// TIA Portal project "SCADA_project" (V15.1)

(* hardware
DEVICE "S7300/ET200M station_1"  S7-300 station
   slot 0: "Rail_0"  Rail  6ES7 390-1***0-0AA0
   slot 1: "PS 307 10A_1"  PS 307 10A  6ES7 307-1KA02-0AA0
   slot 2: "PLC_1"  CPU 315-2 PN/DP  6ES7 315-2EH14-0AB0  V3.2
      slot 2: "PROFINET interface_1"  PN-IO
         slot 1: "Port_1"  Port
         slot 2: "Port_2"  Port
   slot 4: "DI 16x24VDC_1"  DI16 x 24VDC  6ES7 321-1BH02-0AA0
   slot 5: "DO 16x24VDC/0.5A_1"  DO16 x 24VDC / 0.5A  6ES7 322-1BH01-0AA0
   slot 6: "AI 8x16BIT_1"  AI8 x 16 bits  6ES7 331-7NF00-0AB0
DEVICE "PC-System_2"  SIMATIC PC station
   slot 0: "SIMATIC PC station"  Rail  SIMATIC PC-Station  V1.0
      slot 125: "Stationmanager"  Station_Manager  V6.0.4
   slot 1: "HMI_RT_2"  WinCC RT Advanced  6AV2 104-0xxxx-xxxx  15.1.0.0
      slot 33792: "Host interface"  Host interface
   slot 2: "IE general_1"  IE General  IE_CP  V8.2.0
*)

// ===== PLC "PLC_1"  CPU 315-2 PN/DP =====

VAR_GLOBAL   // PLC tag table "Default tag table"
   "LT140" AT %ID0 : Real;   // Level transmitter T140
   "LT150" AT %ID4 : Real;   // Level transmitter T150
   "LT160" AT %ID8 : Real;   // Level transmitter T160
   "LT170" AT %ID12 : Real;   // Level transmitter T170
   "Pump100A_start" AT %M0.0 : Bool;   // Pump
   "Pump100A_stop" AT %M0.1 : Bool;   // Pump
   "Pump770A_start" AT %M0.2 : Bool;   // Pump
   "Pump770A_stop" AT %M0.3 : Bool;   // Pump
   "Pump771A_start" AT %M0.4 : Bool;   // Pump
   "Pump771A_stop" AT %M0.5 : Bool;   // Pump
   "Pump100A" AT %Q4.0 : Bool;
   "Pump770A" AT %Q4.1 : Bool;
   "Pump771A" AT %Q4.2 : Bool;
   "SV1401_open" AT %M0.6 : Bool;
   "SV1401_close" AT %M0.7 : Bool;
   "SV1501_open" AT %M1.0 : Bool;
   "SV1501_close" AT %M1.1 : Bool;
   "SV1601_open" AT %M1.2 : Bool;
   "SV1601_close" AT %M1.3 : Bool;
   "SV1402_open" AT %M1.4 : Bool;
   "SV1402_close" AT %M1.5 : Bool;
   "SV1502_open" AT %M1.6 : Bool;
   "SV1502_close" AT %M1.7 : Bool;
   "SV1602_open" AT %M2.0 : Bool;
   "SV1602_close" AT %M2.1 : Bool;
   "SV1701_open" AT %M2.2 : Bool;
   "SV1701_close" AT %M2.3 : Bool;
   "SV1702_open" AT %M2.4 : Bool;
   "SV1702_close" AT %M2.5 : Bool;
   "SV1401" AT %Q4.3 : Bool;
   "SV1501" AT %Q4.4 : Bool;
   "SV1601" AT %Q4.5 : Bool;
   "SV1701" AT %Q4.6 : Bool;
   "SV1402" AT %Q4.7 : Bool;
   "SV1502" AT %Q5.0 : Bool;
   "SV1602" AT %Q5.1 : Bool;
   "SV1702" AT %Q5.2 : Bool;
   "H_alarm_140" AT %Q5.3 : Bool;
   "L_alarm_140" AT %Q5.4 : Bool;
   "H_alarm_150" AT %Q5.5 : Bool;
   "L_alarm_150" AT %Q5.6 : Bool;
   "H_alarm_160" AT %Q5.7 : Bool;
   "L_alarm_160" AT %Q6.0 : Bool;
   "H_alarm_170" AT %Q6.1 : Bool;
   "L_alarm_170" AT %Q6.2 : Bool;
   "Tank_140_cur_vol" AT %MD5 : Real;
   "Tank_150_cur_vol" AT %MD10 : Real;
   "Tank_160_cur_vol" AT %MD14 : Real;
   "Tank_170_cur_vol" AT %MD18 : Real;
   "dis_alarm_tag" AT %MW48 : Int;
END_VAR

VAR_GLOBAL CONSTANT   // PLC tag table "Default tag table"
   "Tank140_volume" : Real := 1500.0;
   "Tank140_h_alarm_val" : Real := 1350.0;
   "Tank150_volume" : Real := 2500.0;
   "Tank150_h_alarm_val" : Real := 2250.0;
   "Tank160_volume" : Real := 3000.0;
   "Tank160_h_alarm_val" : Real := 2700.0;
   "Tank170_volume" : Real := 10000.0;
   "Tank170_h_alarm_val" : Real := 9000.0;
   "usersss" : Int := 5;
END_VAR

VAR_GLOBAL   // PLC tag table "User Variables"
   "tank_140_capacity" AT %MD0 : Real;
   "tank_140_high_limit" AT %MD4 : Real;
   "tank_140_low_limit" AT %MD8 : Real;
   "tank_150_capacity" AT %MD12 : Real;
   "tank_150_high_limit" AT %MD16 : Real;
   "tank_150_low_limit" AT %MD20 : Real;
   "tank_160_capacity" AT %MD24 : Real;
   "tank_160_high_limit" AT %MD28 : Real;
   "tank_160_low_limit" AT %MD32 : Real;
   "tank_170_capacity" AT %MD36 : Real;
   "tank_170_high_limit" AT %MD40 : Real;
   "tank_170_low_limit" AT %MD44 : Real;
END_VAR

DATA_BLOCK "FP_Dtabase"   // DB1
{ S7_Optimized_Access := 'FALSE' }
VERSION : 0.1
   VAR
      Pump100A_visibility : Bool := true;
      Pump100A_tag_name : String := 'Pump100A FP';
      Pump770A_visibility : Bool := true;
      Pump770A_tag_name : String := 'Pump770A FP';
      Pump771A_visibility : Bool := true;
      Pump771A_tag_name : String := 'Pump771A FP';
      SV1401_visibility : Bool := true;
      SV1401_tag_name : String := 'SV1401 FP';
      SV1402_visibility : Bool := true;
      SV1402_tag_name : String := 'SV1402 FP';
      SV1501_visibility : Bool := true;
      SV1501_tag_name : String := 'SV1501 FP';
      SV1502_visibility : Bool := true;
      SV1502_tag_name : String := 'SV1502 FP';
      SV1601_visibility : Bool := true;
      SV1601_tag_name : String := 'SV1601 FP';
      SV1602_visibility : Bool := true;
      SV1602_tag_name : String := 'SV1602 FP';
      SV1701_visibility : Bool := true;
      SV1701_tag_name : String := 'SV1701 FP';
      SV1702_visibility : Bool := true;
      SV1702_tag_name : String := 'SV1702 FP';
   END_VAR
BEGIN
END_DATA_BLOCK

DATA_BLOCK "my_variables_db"   // DB2
{ S7_Optimized_Access := 'FALSE' }
VERSION : 0.1
   VAR
      tank_140_int_cap : Int := 1500;
      tank_150_int_cap : Int := 2500;
      tank_160_int_cap : Int := 3000;
      tank_170_int_cap : Int := 10000;
      zero : Int := 0;
      user_name_txt : String := 'Username';
      group_no_txt : String := 'Group No';
   END_VAR
BEGIN
END_DATA_BLOCK

FUNCTION "SV1x01" : Void   // FC1, SCL
{ S7_Optimized_Access := 'FALSE' }
VERSION : 0.1
   VAR_INPUT
      Open_valve : Bool;
      Close_valve : Bool;
      High_alarm : Bool;
      Low_alarm : Bool;
      SV1x02 : Bool;
   END_VAR
   VAR_IN_OUT
      SV1x1 : Bool;
   END_VAR
BEGIN

   (* The inlet valve should be opened in case 
   Open Valve command is receieved or Low alarm
   of the corresponding tank is active *)
   IF #Open_valve OR #Low_alarm THEN
       #SV1x1 := TRUE;

   (* The inlet valve should be closed in case 
   Close Valve command is receieved 
   or High alarm of the corresponding tank is active. 
   Additionally, it creates an interlock between SV1x02/01 *)
   ELSIF #High_alarm OR #Close_valve OR #SV1x02 THEN
       #SV1x1 := FALSE;
   END_IF;
END_FUNCTION

FUNCTION "TankAlarm" : Void   // FC2, SCL
{ S7_Optimized_Access := 'FALSE' }
VERSION : 0.1
   VAR_INPUT
      High_alarm_limit : Real;
      Low_alarm_limit : Real;
      Tank_vol : Real;
   END_VAR
   VAR_IN_OUT
      High_alarm : Bool;
      Low_alarm : Bool;
   END_VAR
BEGIN
   #Low_alarm := False;
   #High_alarm := False;

   (*Activate alarms according to the scaled volume*)
   IF #Tank_vol >= #High_alarm_limit THEN
     #High_alarm := TRUE;
   ELSIF #Tank_vol <= #Low_alarm_limit THEN
     #Low_alarm := TRUE;
   END_IF;
END_FUNCTION

FUNCTION "my_scaler_function" : Void   // FC3, SCL
{ S7_Optimized_Access := 'FALSE' }
VERSION : 0.1
   VAR_INPUT
      IN_1_MIN : Real;
      IN_1_MAX : Real;
      IN_2_MIN : Real;
      IN_2_MAX : Real;
      Real_value : Real;
   END_VAR
   VAR_IN_OUT
      my_scaler_function : Real;
   END_VAR
BEGIN
   #my_scaler_function := (#IN_2_MAX - #IN_2_MIN) / (#IN_1_MAX - #IN_1_MIN) * (#Real_value - #IN_1_MIN) + #IN_2_MIN;
   (*Function to scale the level transmitter output signal*)
END_FUNCTION

FUNCTION "Pump100A_func" : Void   // FC4, SCL
{ S7_Optimized_Access := 'FALSE' }
VERSION : 0.1
   VAR_INPUT
      Start_pump : Bool;
      Stop_pump : Bool;
      L_alarm_140 : Bool;
      L_alarm_150 : Bool;
      L_alarm_160 : Bool;
   END_VAR
   VAR_IN_OUT
      Pump100A_func : Bool;
      SV1401 : Bool;
      SV1501 : Bool;
      SV1601 : Bool;
   END_VAR
BEGIN

   (*If at least one Slave Inlet Valve is open AND Start Pump command was recieved OR*)
   IF ((#SV1401 OR #SV1501 OR #SV1601) AND #Start_pump)
       (*OR If at least one Slave Tank has active Low Alarm then Start the Pump100A*)
       OR (#L_alarm_140 OR #L_alarm_150 OR #L_alarm_160) THEN
       #Pump100A_func := TRUE;
   END_IF;

   (*Don not allow to operate Pump100A unless at least one Slave Inlet valve is open*)
   IF NOT (#SV1401 OR #SV1501 OR #SV1601) THEN
       #Pump100A_func := FALSE;
   END_IF;

   (*In case stop pump command was recieved stop pump and close all slave inlet valves*)
   IF #Stop_pump THEN
       #Pump100A_func := FALSE;
       #SV1401 := FALSE;
       #SV1501 := FALSE;
       #SV1601 := FALSE;
   END_IF;
END_FUNCTION

FUNCTION "SV1x02" : Void   // FC5, SCL
{ S7_Optimized_Access := 'FALSE' }
VERSION : 0.1
   VAR_INPUT
      Close_valve : Bool;
      Open_valve : Bool;
      High_alarm : Bool;
      Low_alarm : Bool;
   END_VAR
   VAR_IN_OUT
      SV1x02 : Bool;
   END_VAR
BEGIN

   (*If Open Valve command was recieved, 
   it will be opened*)

   IF #Open_valve THEN
       #SV1x02 := TRUE;

   (* When Close Valce command was recieved OR
    Low alarm of the corresponding tank is active
   then its outlet valve should be closed*)
   ELSIF #Close_valve OR #Low_alarm THEN
       #SV1x02 := FALSE;
   END_IF;
END_FUNCTION

FUNCTION "Pump770A_func" : Void   // FC6, SCL
{ S7_Optimized_Access := 'FALSE' }
VERSION : 0.1
   VAR_INPUT
      H_alarm_170 : Bool;
      L_alarm_170 : Bool;
      SV1701 : Bool;
      L_alarm_140 : Bool;
      L_alarm_150 : Bool;
      L_alarm_160 : Bool;
      SV1401 : Bool;
      SV1501 : Bool;
      SV1601 : Bool;
      Pump100A : Bool;
      Start_pump : Bool;
      Stop_pump : Bool;
   END_VAR
   VAR_IN_OUT
      SV1402 : Bool;
      SV1502 : Bool;
      SV1602 : Bool;
      Pump770A_func : Bool;
   END_VAR
   VAR_TEMP
      L_alarm_arr : Array[0..3] of Bool;
      SV1x02_arr : Array[0..3] of Bool;
      i : Int;
      flag_avaiable_tank : Bool;
   END_VAR
BEGIN
   (* Fill a temporary allocated array with Low alarm and 
   outlet valvestatus of the slave tanks. Due to its convenience, 
   iterational method was implemented*)

   #L_alarm_arr[0] := #L_alarm_140;
   #L_alarm_arr[1] := #L_alarm_150;
   #L_alarm_arr[2] := #L_alarm_160;

   #SV1x02_arr[0] := #SV1402;
   #SV1x02_arr[1] := #SV1502;
   #SV1x02_arr[2] := #SV1602;


   #i := 0; (* Counter for the iteration*)
   #flag_avaiable_tank := FALSE; (*It will be TRUE if any of slave outlet valve is open*)

   (*If there is no enough product in the master tank OR
     Start Pump770A command was recieved AND Tank is not full AND Inlet valve is open
     search for the avilable** slave tank(s) to fill the master tank*)
   IF #L_alarm_170 THEN
       REPEAT
           (* **If a slave tank has enough product (NOT Low alarm)
             then use it to fill the master tank*)
           IF NOT #L_alarm_arr[#i] THEN
               #SV1x02_arr[#i] := TRUE;
               #flag_avaiable_tank := TRUE;
           END_IF;
           #i := #i + 1;
       UNTIL (#i = 3)
       END_REPEAT;

       (*Start tank only if at least one slave tank is available*)
       #Pump770A_func := #flag_avaiable_tank;
   END_IF;

   (*Manual Control for Pump77A*)
   #i := 0;
   IF (NOT #H_alarm_170 AND #Start_pump AND #SV1701) THEN
       REPEAT
           IF #SV1x02_arr[#i] THEN
               #flag_avaiable_tank := TRUE;
           END_IF;
           #i := #i + 1;
       UNTIL (#i = 3)
       END_REPEAT;
       #Pump770A_func := #flag_avaiable_tank;
   END_IF;


   #i := 0;

   (* If Master tank is full OR There's not available slave tank*)
   IF #H_alarm_170 OR #Stop_pump OR NOT (#SV1x02_arr[0] OR #SV1x02_arr[1] OR #SV1x02_arr[2]) THEN
       (*Stop Pump770A and all slave outlet valves*)
       #Pump770A_func := FALSE;
       "SV1701" := FALSE;

       REPEAT
           #SV1x02_arr[#i] := FALSE;
           #i := #i + 1;
       UNTIL (#i = 3)
       END_REPEAT;
   END_IF;

   (*Update status of slave outlet valves regarding the recent computation*)
   #SV1402 := #SV1x02_arr[0];
   #SV1502 := #SV1x02_arr[1];
   #SV1602 := #SV1x02_arr[2];
END_FUNCTION

FUNCTION "SV1701_func" : Void   // FC7, SCL
{ S7_Optimized_Access := 'FALSE' }
VERSION : 0.1
   VAR_INPUT
      Open_valve : Bool;
      Close_valve : Bool;
      High_alarm : Bool;
      L_alarm_170 : Bool;
      Pump770A : Bool;
   END_VAR
   VAR_IN_OUT
      SV1701_func : Bool;
   END_VAR
BEGIN

   (*IF Open Valve command recieved Open the inlet valve
   and as an interlock Close and Power off the 
   outlet valve and Pump771A*)
   IF #Open_valve THEN
       #SV1701_func := TRUE;
       "Pump771A" := FALSE;
       "SV1702" := FALSE;
   END_IF;

   (*In case Low alarm activated AND Pump770A should be activated
   then Open the inlet valve*)
   IF #L_alarm_170 AND #Pump770A THEN
       #SV1701_func := TRUE;
   END_IF;

   (*If High alarm is activate O CMD of Closing the inlet valve was receievd
   Close the Inlet valve*)
   IF #High_alarm OR #Close_valve THEN
       #SV1701_func := FALSE;
   END_IF;
END_FUNCTION

FUNCTION "SV1702_func" : Void   // FC8, SCL
{ S7_Optimized_Access := 'FALSE' }
VERSION : 0.1
   VAR_INPUT
      Close_valve : Bool;
      Open_valve : Bool;
      High_alarm : Bool;
      Low_alarm : Bool;
   END_VAR
   VAR_IN_OUT
      SV1702_func : Bool;
      SV1701 : Bool;
   END_VAR
BEGIN
   (* If Open valve command was recieved AND Low alarm is not active
    Close all Slave Outlet and Master Inlet Valves, Stop Pump770 and Open the Outlet Valve*)
   IF #Open_valve AND NOT #Low_alarm THEN
       #SV1702_func := TRUE;
       #SV1701 := FALSE;

       "SV1402" := FALSE;
       "SV1502" := FALSE;
       "SV1602" := FALSE;

       "Pump770A" := FALSE;

   (*If Close valve command was recieved OR there's no enough
   product in the tank (Low alarm is active) close the outlet valve *)
   ELSIF #Close_valve OR  #Low_alarm  THEN
       #SV1702_func := FALSE;
       "Pump771A" := FALSE;
   END_IF;
END_FUNCTION

FUNCTION "Pump771_func" : Void   // FC9, SCL
{ S7_Optimized_Access := 'FALSE' }
VERSION : 0.1
   VAR_INPUT
      Start_pump : Bool;
      Stop_pump : Bool;
   END_VAR
   VAR_IN_OUT
      Pump771_func : Bool;
      SV1702 : Bool;
   END_VAR
BEGIN

   (* If start Pump771A was recieved AND 
   Outlet valve is open then allow to operate Pump771A*)
   IF #Start_pump AND #SV1702 THEN
       #Pump771_func := TRUE;
   END_IF;

   (*If Pump is operating and Stop command recieved
   Stop the pump and close the outlet valve*)
   IF #Pump771_func AND #Stop_pump THEN
       #Pump771_func := False;
       #SV1702 := FALSE;
   END_IF;
END_FUNCTION

ORGANIZATION_BLOCK "Main"   // OB1, FBD
TITLE = "Main Program Sweep (Cycle)"
{ S7_Optimized_Access := 'FALSE' }
VERSION : 0.1
   VAR_TEMP
      OB1_EV_CLASS : Byte;   // Bits 0-3 = 1 (Coming event), Bits 4-7 = 1 (Event class 1)
      OB1_SCAN_1 : Byte;   // 1 (Cold restart scan 1 of OB 1), 3 (Scan 2-n of OB 1)
      OB1_PRIORITY : Byte;   // Priority of OB Execution
      OB1_OB_NUMBR : Byte;   // 1 (Organization block 1, OB1)
      OB1_RESERVED_1 : Byte;   // Reserved for system
      OB1_RESERVED_2 : Byte;   // Reserved for system
      OB1_PREV_CYCLE : Int;   // Cycle time of previous OB1 scan (milliseconds)
      OB1_MIN_CYCLE : Int;   // Minimum cycle time of OB1 (milliseconds)
      OB1_MAX_CYCLE : Int;   // Maximum cycle time of OB1 (milliseconds)
      OB1_DATE_TIME : Date_And_Time;   // Date and time OB1 started
   END_VAR
BEGIN

REGION Network 1
   // Pump100A
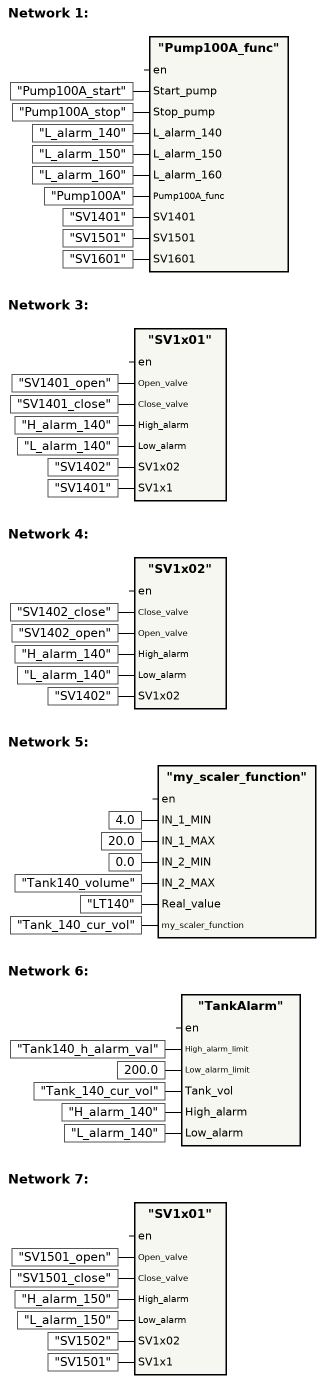
   "Pump100A_func"(Start_pump := "Pump100A_start",
                   Stop_pump := "Pump100A_stop",
                   L_alarm_140 := "L_alarm_140",
                   L_alarm_150 := "L_alarm_150",
                   L_alarm_160 := "L_alarm_160",
                   Pump100A_func := "Pump100A",
                   SV1401 := "SV1401",
                   SV1501 := "SV1501",
                   SV1601 := "SV1601");
END_REGION

REGION Network 3
   // Tank 140
   "SV1x01"(Open_valve := "SV1401_open",
            Close_valve := "SV1401_close",
            High_alarm := "H_alarm_140",
            Low_alarm := "L_alarm_140",
            SV1x02 := "SV1402",
            SV1x1 := "SV1401");
END_REGION

REGION Network 4
   "SV1x02"(Close_valve := "SV1402_close",
            Open_valve := "SV1402_open",
            High_alarm := "H_alarm_140",
            Low_alarm := "L_alarm_140",
            SV1x02 := "SV1402");
END_REGION

REGION Network 5
   "my_scaler_function"(IN_1_MIN := 4.0,
                        IN_1_MAX := 20.0,
                        IN_2_MIN := 0.0,
                        IN_2_MAX := "Tank140_volume",
                        Real_value := "LT140",
                        my_scaler_function := "Tank_140_cur_vol");
END_REGION

REGION Network 6
   "TankAlarm"(High_alarm_limit := "Tank140_h_alarm_val",
               Low_alarm_limit := 200.0,
               Tank_vol := "Tank_140_cur_vol",
               High_alarm := "H_alarm_140",
               Low_alarm := "L_alarm_140");
END_REGION

REGION Network 7
   // Tank 150
   "SV1x01"(Open_valve := "SV1501_open",
            Close_valve := "SV1501_close",
            High_alarm := "H_alarm_150",
            Low_alarm := "L_alarm_150",
            SV1x02 := "SV1502",
            SV1x1 := "SV1501");
END_REGION

REGION Network 8
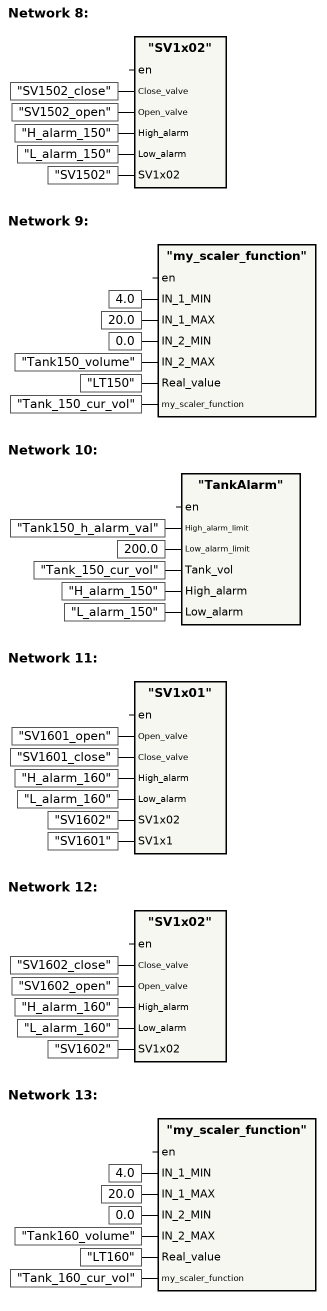
   "SV1x02"(Close_valve := "SV1502_close",
            Open_valve := "SV1502_open",
            High_alarm := "H_alarm_150",
            Low_alarm := "L_alarm_150",
            SV1x02 := "SV1502");
END_REGION

REGION Network 9
   "my_scaler_function"(IN_1_MIN := 4.0,
                        IN_1_MAX := 20.0,
                        IN_2_MIN := 0.0,
                        IN_2_MAX := "Tank150_volume",
                        Real_value := "LT150",
                        my_scaler_function := "Tank_150_cur_vol");
END_REGION

REGION Network 10
   "TankAlarm"(High_alarm_limit := "Tank150_h_alarm_val",
               Low_alarm_limit := 200.0,
               Tank_vol := "Tank_150_cur_vol",
               High_alarm := "H_alarm_150",
               Low_alarm := "L_alarm_150");
END_REGION

REGION Network 11
   // Tank 160
   "SV1x01"(Open_valve := "SV1601_open",
            Close_valve := "SV1601_close",
            High_alarm := "H_alarm_160",
            Low_alarm := "L_alarm_160",
            SV1x02 := "SV1602",
            SV1x1 := "SV1601");
END_REGION

REGION Network 12
   "SV1x02"(Close_valve := "SV1602_close",
            Open_valve := "SV1602_open",
            High_alarm := "H_alarm_160",
            Low_alarm := "L_alarm_160",
            SV1x02 := "SV1602");
END_REGION

REGION Network 13
   "my_scaler_function"(IN_1_MIN := 4.0,
                        IN_1_MAX := 20.0,
                        IN_2_MIN := 0.0,
                        IN_2_MAX := "Tank160_volume",
                        Real_value := "LT160",
                        my_scaler_function := "Tank_160_cur_vol");
END_REGION

REGION Network 14
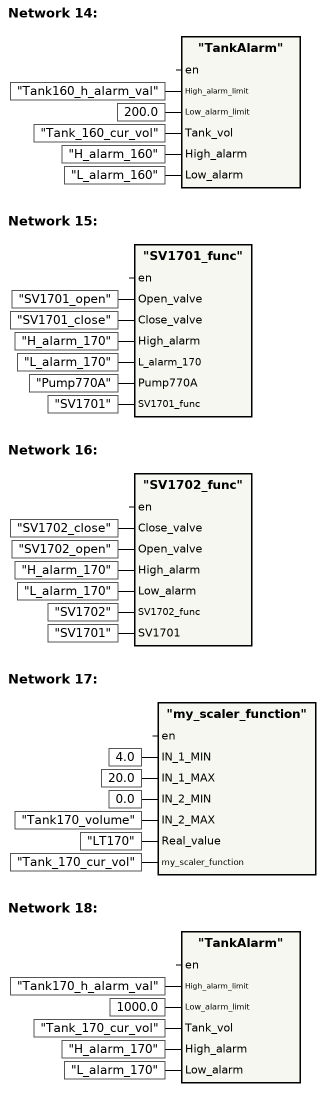
   "TankAlarm"(High_alarm_limit := "Tank160_h_alarm_val",
               Low_alarm_limit := 200.0,
               Tank_vol := "Tank_160_cur_vol",
               High_alarm := "H_alarm_160",
               Low_alarm := "L_alarm_160");
END_REGION

REGION Network 15
   // Tank 170
   "SV1701_func"(Open_valve := "SV1701_open",
                 Close_valve := "SV1701_close",
                 High_alarm := "H_alarm_170",
                 L_alarm_170 := "L_alarm_170",
                 Pump770A := "Pump770A",
                 SV1701_func := "SV1701");
END_REGION

REGION Network 16
   "SV1702_func"(Close_valve := "SV1702_close",
                 Open_valve := "SV1702_open",
                 High_alarm := "H_alarm_170",
                 Low_alarm := "L_alarm_170",
                 SV1702_func := "SV1702",
                 SV1701 := "SV1701");
END_REGION

REGION Network 17
   "my_scaler_function"(IN_1_MIN := 4.0,
                        IN_1_MAX := 20.0,
                        IN_2_MIN := 0.0,
                        IN_2_MAX := "Tank170_volume",
                        Real_value := "LT170",
                        my_scaler_function := "Tank_170_cur_vol");
END_REGION

REGION Network 18
   "TankAlarm"(High_alarm_limit := "Tank170_h_alarm_val",
               Low_alarm_limit := 1000.0,
               Tank_vol := "Tank_170_cur_vol",
               High_alarm := "H_alarm_170",
               Low_alarm := "L_alarm_170");
END_REGION

REGION Network 19
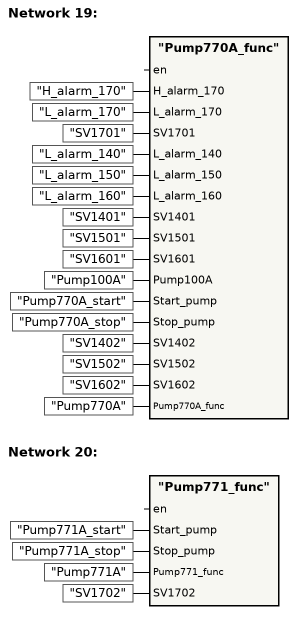
   "Pump770A_func"(H_alarm_170 := "H_alarm_170",
                   L_alarm_170 := "L_alarm_170",
                   SV1701 := "SV1701",
                   L_alarm_140 := "L_alarm_140",
                   L_alarm_150 := "L_alarm_150",
                   L_alarm_160 := "L_alarm_160",
                   SV1401 := "SV1401",
                   SV1501 := "SV1501",
                   SV1601 := "SV1601",
                   Pump100A := "Pump100A",
                   Start_pump := "Pump770A_start",
                   Stop_pump := "Pump770A_stop",
                   SV1402 := "SV1402",
                   SV1502 := "SV1502",
                   SV1602 := "SV1602",
                   Pump770A_func := "Pump770A");
END_REGION

REGION Network 20
   "Pump771_func"(Start_pump := "Pump771A_start",
                  Stop_pump := "Pump771A_stop",
                  Pump771_func := "Pump771A",
                  SV1702 := "SV1702");
END_REGION
END_ORGANIZATION_BLOCK

(* ===== HMI "HMI_RT_2" =====
system functions are stored by id; their names below are inferred from use
connection "HMI_Connection_1": ETHERNET, SIMATIC S7 300/400 MPI

HMI tags "Default tag table"
   "Tag_ScreenNumber" : UInt, internal
   "Current_user" : WString[10], internal
   "Pump100A" : Bool = PLC Pump100A AT %Q4.0, 1 s
   "SV1401" : Bool = PLC SV1401 AT %Q4.3, 1 s
   "SV1402" : Bool = PLC SV1402 AT %Q4.7, 1 s
   "SV1501" : Bool = PLC SV1501 AT %Q4.4, 1 s
   "SV1502" : Bool = PLC SV1502 AT %Q5.0, 1 s
   "SV1601" : Bool = PLC SV1601 AT %Q4.5, 1 s
   "SV1602" : Bool = PLC SV1602 AT %Q5.1, 1 s
   "Pump770A" : Bool = PLC Pump770A AT %Q4.1, 1 s
   "Pump771A" : Bool = PLC Pump771A AT %Q4.2, 1 s
   "SV1701" : Bool = PLC SV1701 AT %Q4.6, 1 s
   "SV1702" : Bool = PLC SV1702 AT %Q5.2, 1 s
   "FP_Dtabase_Pump100A_visibility" : Bool = PLC FP_Dtabase.Pump100A_visibility AT %DB1.DBX0.0, 1 s
   "Pump100A_start" : Bool = PLC Pump100A_start AT %M0.0, 1 s
   "Pump100A_stop" : Bool = PLC Pump100A_stop AT %M0.1, 1 s
   "FP_Dtabase_Pump100A_tag_name" : String[254] = PLC FP_Dtabase.Pump100A_tag_name AT %DB1.DBX2.0, 1 s
   "SV1401_close" : Bool = PLC SV1401_close AT %M0.7, 1 s
   "FP_Dtabase_SV1401_visibility" : Bool = PLC FP_Dtabase.SV1401_visibility AT %DB1.DBX774.0, 1 s
   "SV1401_open" : Bool = PLC SV1401_open AT %M0.6, 1 s
   "FP_Dtabase_SV1401_tag_name" : String[254] = PLC FP_Dtabase.SV1401_tag_name AT %DB1.DBX776.0, 1 s
   "Tank_140_vol" : Real = PLC Tank_140_cur_vol AT %MD5, 1 s
   "L_alarm_140" : Bool = PLC L_alarm_140 AT %Q5.4, 1 s
   "H_alarm_140" : Bool = PLC H_alarm_140 AT %Q5.3, 1 s
   "SV1402_close" : Bool = PLC SV1402_close AT %M1.5, 1 s
   "FP_Dtabase_SV1402_visibility" : Bool = PLC FP_Dtabase.SV1402_visibility AT %DB1.DBX1032.0, 1 s
   "SV1402_open" : Bool = PLC SV1402_open AT %M1.4, 1 s
   "FP_Dtabase_SV1402_tag_name" : String[254] = PLC FP_Dtabase.SV1402_tag_name AT %DB1.DBX1034.0, 1 s
   "FP_Dtabase_Pump770A_visibility" : Bool = PLC FP_Dtabase.Pump770A_visibility AT %DB1.DBX258.0, 1 s
   "Pump770A_start" : Bool = PLC Pump770A_start AT %M0.2, 1 s
   "Pump770A_stop" : Bool = PLC Pump770A_stop AT %M0.3, 1 s
   "FP_Dtabase_Pump770A_tag_name" : String[254] = PLC FP_Dtabase.Pump770A_tag_name AT %DB1.DBX260.0, 1 s
   "SV1501_close" : Bool = PLC SV1501_close AT %M1.1, 1 s
   "SV1501_open" : Bool = PLC SV1501_open AT %M1.0, 1 s
   "FP_Dtabase_SV1501_visibility" : Bool = PLC FP_Dtabase.SV1501_visibility AT %DB1.DBX1290.0, 1 s
   "FP_Dtabase_SV1501_tag_name" : String[254] = PLC FP_Dtabase.SV1501_tag_name AT %DB1.DBX1292.0, 1 s
   "SV1502_close" : Bool = PLC SV1502_close AT %M1.7, 1 s
   "SV1502_open" : Bool = PLC SV1502_open AT %M1.6, 1 s
   "FP_Dtabase_SV1502_visibility" : Bool = PLC FP_Dtabase.SV1502_visibility AT %DB1.DBX1548.0, 1 s
   "FP_Dtabase_SV1502_tag_name" : String[254] = PLC FP_Dtabase.SV1502_tag_name AT %DB1.DBX1550.0, 1 s
   "H_alarm_150" : Bool = PLC H_alarm_150 AT %Q5.5, 1 s
   "L_alarm_150" : Bool = PLC L_alarm_150 AT %Q5.6, 1 s
   "Tank_150_cur_vol" : Real = PLC Tank_150_cur_vol AT %MD10, 1 s
   "SV1601_close" : Bool = PLC SV1601_close AT %M1.3, 1 s
   "SV1601_open" : Bool = PLC SV1601_open AT %M1.2, 1 s
   "FP_Dtabase_SV1601_visibility" : Bool = PLC FP_Dtabase.SV1601_visibility AT %DB1.DBX1806.0, 1 s
   "FP_Dtabase_SV1601_tag_name" : String[254] = PLC FP_Dtabase.SV1601_tag_name AT %DB1.DBX1808.0, 1 s
   "SV1602_close" : Bool = PLC SV1602_close AT %M2.1, 1 s
   "SV1602_open" : Bool = PLC SV1602_open AT %M2.0, 1 s
   "FP_Dtabase_SV1602_visibility" : Bool = PLC FP_Dtabase.SV1602_visibility AT %DB1.DBX2064.0, 1 s
   "FP_Dtabase_SV1602_tag_name" : String[254] = PLC FP_Dtabase.SV1602_tag_name AT %DB1.DBX2066.0, 1 s
   "Tank_160_cur_vol" : Real = PLC Tank_160_cur_vol AT %MD14, 1 s
   "H_alarm_160" : Bool = PLC H_alarm_160 AT %Q5.7, 1 s
   "L_alarm_160" : Bool = PLC L_alarm_160 AT %Q6.0, 1 s
   "tank_160_capacity" : Real = PLC tank_160_capacity AT %MD24, 1 s
   "my_variables_db_tank_140_int_cap" : Int = PLC my_variables_db.tank_140_int_cap AT %DB2.DBW0, 1 s
   "my_variables_db_zero" : Int = PLC my_variables_db.zero AT %DB2.DBW8, 1 s
   "my_variables_db_tank_160_int_cap" : Int = PLC my_variables_db.tank_160_int_cap AT %DB2.DBW4, 1 s
   "my_variables_db_tank_150_int_cap" : Int = PLC my_variables_db.tank_150_int_cap AT %DB2.DBW2, 1 s
   "tank_150_capacity" : Real = PLC tank_150_capacity AT %MD12, 1 s
   "Tank_170_cur_vol" : Real = PLC Tank_170_cur_vol AT %MD18, 1 s
   "H_alarm_170" : Bool = PLC H_alarm_170 AT %Q6.1, 1 s
   "L_alarm_170" : Bool = PLC L_alarm_170 AT %Q6.2, 1 s
   "my_variables_db_tank_170_int_cap" : Int = PLC my_variables_db.tank_170_int_cap AT %DB2.DBW6, 1 s
   "SV1701_close" : Bool = PLC SV1701_close AT %M2.3, 1 s
   "SV1701_open" : Bool = PLC SV1701_open AT %M2.2, 1 s
   "FP_Dtabase_SV1701_visibility" : Bool = PLC FP_Dtabase.SV1701_visibility AT %DB1.DBX2322.0, 1 s
   "FP_Dtabase_SV1701_tag_name" : String[254] = PLC FP_Dtabase.SV1701_tag_name AT %DB1.DBX2324.0, 1 s
   "SV1702_close" : Bool = PLC SV1702_close AT %M2.5, 1 s
   "SV1702_open" : Bool = PLC SV1702_open AT %M2.4, 1 s
   "FP_Dtabase_SV1702_visibility" : Bool = PLC FP_Dtabase.SV1702_visibility AT %DB1.DBX2580.0, 1 s
   "FP_Dtabase_SV1702_tag_name" : String[254] = PLC FP_Dtabase.SV1702_tag_name AT %DB1.DBX2582.0, 1 s
   "Pump771A_start" : Bool = PLC Pump771A_start AT %M0.4, 1 s
   "Pump771A_stop" : Bool = PLC Pump771A_stop AT %M0.5, 1 s
   "FP_Dtabase_Pump771A_visibility" : Bool = PLC FP_Dtabase.Pump771A_visibility AT %DB1.DBX516.0, 1 s
   "FP_Dtabase_Pump771A_tag_name" : String[254] = PLC FP_Dtabase.Pump771A_tag_name AT %DB1.DBX518.0, 1 s
   "my_variables_db_user_name_txt" : String[254] = PLC my_variables_db.user_name_txt AT %DB2.DBX10.0, 1 s
   "my_variables_db_group_no_txt" : String[254] = PLC my_variables_db.group_no_txt AT %DB2.DBX266.0, 1 s
   "current_group_no" : Int, internal

discrete alarms
   1: 'Level Transmitter LT140 is faulty / Level transmitter of tank140 doesnot work properly!', class Acknowledgement bit 0
   2: 'Level Transmitter LT150 is faulty / Cause of Alarm: Level Transmitter of Tank150 doesnot work properly! Corrective Actions: Inform Engineers! Consequence of no Action: Cannot control level in the Tank150', class Acknowledgement bit 0
   3: 'SV1401 has failed to close / Cause of Alarm: Inlet SV of Tank140 failed to close! Corrective Actions: Inform Engineers! Consequence of no Action: Empty Tank140', class Errors bit 0
   4: 'SV1501 has failed to close', class Errors bit 0

analog alarms
   1: 'Level is low in Tank140 / Cause of Alarm: Low Level in the Tank140 Corrective Actions: Open inlet SV1401 Consequence of no Action: Empty Tank140', class Errors, trigger "Tank_140_vol"
   2: 'Level is high in Tank140 / Cause of Alarm: High Level in the Tank140 Corrective Actions: Close inlet SV1401 Consequence of no Action: Overfill and Overpressure in Tank140', class Errors, trigger "Tank_140_vol"
   3: 'Level is low in Tank150 / Cause of Alarm: Low Level in the Tank150 Corrective Actions: Open inlet SV1501 Consequence of no Action: Empty Tank150', class Errors, trigger "Tank_150_cur_vol"
   4: 'Level is high in Tank150 / Cause of Alarm: High Level in the Tank150 Corrective Actions: Close inlet SV1501 Consequence of no Action: Overfill and Overpressure in Tank150', class Errors, trigger "Tank_150_cur_vol"
   5: 'Level is low in Tank160 / Cause of Alarm: Low Level in the Tank160 Corrective Actions: Open inlet SV1601 Consequence of no Action: Empty Tank160', class Errors, trigger "Tank_160_cur_vol"
   6: 'Level is high in Tank160 / Cause of Alarm: High Level in the Tank160 Corrective Actions: Close inlet SV1601 Consequence of no Action: Overfill and Overpressure in Tank160', class Errors, trigger "Tank_160_cur_vol"
   7: 'Level is low in Tank170 / Cause of Alarm: Low Level in the Tank170 Corrective Actions: Open inlet SV1701 Consequence of no Action: Empty Tank170', class Errors, trigger "Tank_170_cur_vol"
   8: 'Level is high in Tank170 / Cause of Alarm: High Level in the Tank170 Corrective Actions: Close inlet SV1701 Consequence of no Action: Overfill and Overpressure in Tank170', class Errors, trigger "Tank_170_cur_vol"

text list "Status": 0 'OFF'; 1 'ON'

Template "Template_1" 1980x1078
   AlarmView "Alarm view_Unacknowledged" at 0,0 size 1980x18

screen "TankFarm" 1980x1078, template "Template_1"
   on GenerateScreen: SetTag("Tag_ScreenNumber", 1)
   GraphicView "Graphic view_46" at 1557,132 size 57x129; Picture "Graphic_19"
   GraphicView "Graphic view_45" at 1175,138 size 57x129; Picture "Graphic_19"
   GraphicView "Graphic view_43" at 754,138 size 57x129; Picture "Graphic_19"
   GraphicView "Graphic view_44" at 346,138 size 57x129; Picture "Graphic_19"
   GraphicView "Graphic view_41" at 1427,190 size 327x414; Picture "Graphic_3"
   GraphicView "Graphic view_1" at 250,202 size 251x329; Picture "Graphic_3"
   GraphicView "Graphic view_2" at 290,506 size 76x69; Picture "Graphic_4"
   GraphicView "Graphic view_5" at 301,569 size 83x93; Picture "Graphic_7"
   GraphicView "Graphic view_3" at 290,658 size 76x68; Picture "Graphic_4"
   GraphicView "Graphic view_4" at 383,507 size 76x69; Picture "Graphic_4"
   GraphicView "Graphic view_6" at 394,570 size 83x93; Picture "Graphic_7"
   GraphicView "Graphic view_7" at 383,655 size 76x177; Picture "Graphic_4"
   GraphicView "Graphic view_10" at 658,202 size 251x329; Picture "Graphic_3"
   GraphicView "Graphic view_11" at 698,506 size 76x69; Picture "Graphic_4"
   GraphicView "Graphic view_12" at 709,569 size 83x93; Picture "Graphic_7"
   GraphicView "Graphic view_13" at 698,658 size 76x68; Picture "Graphic_4"
   GraphicView "Graphic view_14" at 791,507 size 76x69; Picture "Graphic_4"
   GraphicView "Graphic view_15" at 802,570 size 83x93; Picture "Graphic_7"
   GraphicView "Graphic view_16" at 791,654 size 76x177; Picture "Graphic_4"
   GraphicView "Graphic view_18" at 572,751 size 128x41; Picture "Graphic_10"
   GraphicView "Graphic view_27" at 440,850 size 795x41; Picture "Graphic_10"
   GraphicView "Graphic view_30" at 784,818 size 91x71; Picture "Graphic_9"
   GraphicView "Graphic view_29" at 397,816 size 94x74; Picture "Graphic_14"
   GraphicView "Graphic view_9" at 164,751 size 965x41; Picture "Graphic_10"
   GraphicView "Graphic view_8" at 285,719 size 91x71; Picture "Graphic_9"
   GraphicView "Graphic view_17" at 692,719 size 91x71; Picture "Graphic_9"
   GraphicView "Graphic view_19" at 1081,202 size 251x329; Picture "Graphic_3"
   GraphicView "Graphic view_20" at 1121,506 size 76x69; Picture "Graphic_4"
   GraphicView "Graphic view_21" at 1132,569 size 83x93; Picture "Graphic_7"
   GraphicView "Graphic view_22" at 1121,658 size 76x66; Picture "Graphic_4"
   GraphicView "Graphic view_23" at 1214,507 size 76x69; Picture "Graphic_4"
   GraphicView "Graphic view_24" at 1225,570 size 83x93; Picture "Graphic_7"
   GraphicView "Graphic view_28" at 1095,717 size 87x74; Picture "Graphic_11"
   GraphicView "Graphic view_25" at 1214,654 size 76x193; Picture "Graphic_4"
   GraphicView "Graphic view_37" at 1491,570 size 76x69; Picture "Graphic_4"
   GraphicView "Graphic view_38" at 1502,633 size 83x93; Picture "Graphic_7"
   GraphicView "Graphic view_39" at 1491,722 size 76x66; Picture "Graphic_4"
   GraphicView "Graphic view_40" at 1466,781 size 87x74; Picture "Graphic_11"
   GraphicView "Graphic view_31" at 1208,818 size 91x71; Picture "Graphic_9"
   GraphicView "Graphic view_35" at 1288,807 size 192x124; Picture "Graphic_16"
   GraphicView "Graphic view_32" at 1612,570 size 76x69; Picture "Graphic_4"
   GraphicView "Graphic view_33" at 1623,633 size 83x93; Picture "Graphic_7"
   GraphicView "Graphic view_34" at 1612,718 size 76x177; Picture "Graphic_4"
   GraphicView "Graphic view_36" at 1626,879 size 94x74; Picture "Graphic_14"
   GraphicView "Graphic view_42" at 1710,870 size 192x124; Picture "Graphic_16"
   GraphicView "Graphic view_26" at 59,742 size 192x124; Picture "Graphic_16"
      Appearance <- "Pump100A"
   Circle "Circle_1" at 127,781 size 48x48
      Appearance <- "Pump100A"
   Rectangle "Rectangle_1" at 317,588 size 23x56
      Appearance <- "SV1401"
   Rectangle "Rectangle_2" at 411,589 size 23x56
      Appearance <- "SV1402"
   Rectangle "Rectangle_3" at 724,588 size 23x56
      Appearance <- "SV1501"
   Rectangle "Rectangle_4" at 820,589 size 23x56
      Appearance <- "SV1502"
   Rectangle "Rectangle_5" at 1150,588 size 23x56
      Appearance <- "SV1601"
   Rectangle "Rectangle_6" at 1244,589 size 23x56
      Appearance <- "SV1602"
   Rectangle "Rectangle_7" at 1519,652 size 23x56
      Appearance <- "SV1701"
   Rectangle "Rectangle_8" at 1640,652 size 23x56
      Appearance <- "SV1702"
   Circle "Circle_2" at 1356,850 size 48x48
      Appearance <- "Pump770A"
   Circle "Circle_3" at 1779,911 size 48x48
      Appearance <- "Pump771A"
   Button "Button_1" at 63,51 size 68x12; TextOff 'Text'
      on Press: ActivateScreen("Main", 0)
   IOField "I/O field_1" at 415,140 size 117x51; FormatPattern 99999
      ProcessValue <- "Tank_140_vol"
   GraphicView "Graphic view_49" at 438,267 size 36x40; Picture "Graphic_20"
      Appearance <- "H_alarm_140"
   GraphicView "Graphic view_50" at 438,448 size 36x40; Picture "Graphic_21"
      Appearance <- "L_alarm_140"
   Bar "Bar_1" at 354,230 size 42x292; MinimumValue 0; MaximumValue 100
      MinimumValue <- "my_variables_db_zero"
      ProcessValue <- "Tank_140_vol"
      MaximumValue <- "my_variables_db_tank_140_int_cap"
   GraphicView "Graphic view_47" at 844,264 size 36x40; Picture "Graphic_20"
      Appearance <- "H_alarm_150"
   GraphicView "Graphic view_48" at 845,445 size 36x40; Picture "Graphic_21"
      Appearance <- "L_alarm_150"
   IOField "I/O field_2" at 828,140 size 117x51; FormatPattern 99999
      ProcessValue <- "Tank_150_cur_vol"
   Bar "Bar_2" at 762,231 size 42x291; MinimumValue 0; MaximumValue 100
      MinimumValue <- "my_variables_db_zero"
      MaximumValue <- "my_variables_db_tank_150_int_cap"
      ProcessValue <- "Tank_150_cur_vol"
   GraphicView "Graphic view_51" at 1266,267 size 36x40; Picture "Graphic_20"
      Appearance <- "H_alarm_160"
   GraphicView "Graphic view_52" at 1265,446 size 36x40; Picture "Graphic_21"
      Appearance <- "L_alarm_160"
   IOField "I/O field_3" at 1247,140 size 117x51; FormatPattern 99999
      ProcessValue <- "Tank_160_cur_vol"
   Bar "Bar_3" at 1186,231 size 42x291; MinimumValue 0; MaximumValue 100
      MinimumValue <- "my_variables_db_zero"
      ProcessValue <- "Tank_160_cur_vol"
      MaximumValue <- "my_variables_db_tank_160_int_cap"
   GraphicView "Graphic view_53" at 1655,274 size 36x40; Picture "Graphic_20"
      Appearance <- "H_alarm_170"
   GraphicView "Graphic view_54" at 1657,509 size 36x40; Picture "Graphic_21"
      Appearance <- "L_alarm_170"
   IOField "I/O field_4" at 1640,136 size 117x51; FormatPattern 99999
      ProcessValue <- "Tank_170_cur_vol"
   Bar "Bar_4" at 1563,226 size 56x366; MinimumValue 0; MaximumValue 100
      MinimumValue <- "my_variables_db_zero"
      MaximumValue <- "my_variables_db_tank_170_int_cap"
      ProcessValue <- "Tank_170_cur_vol"
   Button "Button_2" at 298,91 size 150x35; TextOff 'Tank140'
      on Click: ActivateScreen("Tank140", 0)
   Button "Button_3" at 700,93 size 150x35; TextOff 'Tank150'
      on Click: ActivateScreen("Tank150", 0)
   Button "Button_4" at 1116,91 size 150x35; TextOff 'Tank160'
      on Click: ActivateScreen("Tank160", 0)
   Button "Button_5" at 1505,91 size 150x35; TextOff 'Tank170'
      on Click: ActivateScreen("Tank170", 0)
   Button "Button_7" at 437,258 size 42x67; TextOff 'Text'
      Visibility <- "H_alarm_140"
      on Click: function_efd93a16("hi_alarm_pop_up", 800, 300, -1, -1, 1)
   Button "Button_6" at 1710,33 size 150x35; TextOff 'Trends'
      on Click: ActivateScreen("Trend Screen", 0)
   Button "Button_8" at 436,435 size 42x67; TextOff 'Text'
      on Click: function_efd93a16("lo_alarm_pop_up", 800, 300, -1, -1, 1)
      Visibility <- "L_alarm_140"

screen "Main" 1980x1078
   Button "Button_3" at 712,553 size 478x54; TextOff 'Tank Farm'; Authorization "Operate"
      on Press: ActivateScreen("TankFarm", 0)
   Button "Button_1" at 814,406 size 276x35; TextOff 'Login'
      on Press: function_a2a04561()
   Button "Button_2" at 813,451 size 277x36; TextOff 'Log Out'
      on Press: function_f23ef4c9()
   IOField "I/O field_1" at 953,271 size 136x43; FormatPattern ??????????
      ProcessValue <- "Current_user"
   IOField "I/O field_3" at 814,271 size 136x43; FormatPattern ??????????
      ProcessValue <- "my_variables_db_user_name_txt"
   IOField "I/O field_2" at 953,329 size 136x43; FormatPattern 999
      ProcessValue <- "current_group_no"
   IOField "I/O field_4" at 814,329 size 136x43; FormatPattern ??????????
      ProcessValue <- "my_variables_db_group_no_txt"
   TextField "Text field_1" at 805,166 size 271x34; Text 'Main Screen'
   UserView "User view_1" at 14,677 size 1879x397

screen "Tank140" 1980x1078
   Button "Button_1" at 63,53 size 68x12; TextOff 'Text'
      on Press: ActivateScreen("TankFarm", 0)
   Button "Button_5" at 1185,801 size 155x30; TextOff 'Pump770A FP'
      on Click: ResetBit("FP_Dtabase_Pump770A_visibility")
   Button "Button_4" at 992,558 size 155x30; TextOff 'SV1402 FP'
      on Click: ResetBit("FP_Dtabase_SV1402_visibility")
   Button "Button_3" at 487,557 size 155x30; TextOff 'SV1401 FP'
      on Click: ResetBit("FP_Dtabase_SV1401_visibility")
   Button "Button_2" at 278,766 size 155x30; TextOff 'Pump100A FP'
      on Click: ResetBit("FP_Dtabase_Pump100A_visibility")
   GraphicView "Graphic view_44" at 817,140 size 57x129; Picture "Graphic_19"
   GraphicView "Graphic view_1" at 722,204 size 251x329; Picture "Graphic_3"
   GraphicView "Graphic view_2" at 762,508 size 76x69; Picture "Graphic_4"
   GraphicView "Graphic view_5" at 773,571 size 83x93; Picture "Graphic_7"
   GraphicView "Graphic view_3" at 762,660 size 76x68; Picture "Graphic_4"
   GraphicView "Graphic view_4" at 855,509 size 76x69; Picture "Graphic_4"
   GraphicView "Graphic view_6" at 866,572 size 83x93; Picture "Graphic_7"
   GraphicView "Graphic view_7" at 855,657 size 76x177; Picture "Graphic_4"
   GraphicView "Graphic view_29" at 870,818 size 94x74; Picture "Graphic_14"
   GraphicView "Graphic view_35" at 954,810 size 192x124; Picture "Graphic_16"
   GraphicView "Graphic view_26" at 553,749 size 192x124; Picture "Graphic_16"
      Appearance <- "Pump100A"
   Circle "Circle_1" at 619,788 size 48x48
      Appearance <- "Pump100A"
   Rectangle "Rectangle_1" at 789,590 size 23x56
      Appearance <- "SV1401"
   Rectangle "Rectangle_2" at 883,591 size 23x56
      Appearance <- "SV1402"
   Circle "Circle_2" at 1022,853 size 48x48
      Appearance <- "Pump770A"
   GraphicView "Graphic view_28" at 736,723 size 87x74; Picture "Graphic_11"
   TextField "Text field_1" at 641,8 size 740x90; Text 'Tank 140'
   Group "Group" at 23,35 size 108x47
   IOField "I/O field_1" at 894,145 size 117x51; FormatPattern 99999
      ProcessValue <- "Tank_140_vol"
   GraphicView "Graphic view_49" at 909,283 size 36x40; Picture "Graphic_20"
      Appearance <- "H_alarm_140"
   GraphicView "Graphic view_50" at 911,450 size 36x40; Picture "Graphic_21"
      Appearance <- "L_alarm_140"
   Bar "Bar_1" at 827,253 size 42x271; MinimumValue 0; MaximumValue 100
      MinimumValue <- "my_variables_db_zero"
      MaximumValue <- "my_variables_db_tank_140_int_cap"
      ProcessValue <- "Tank_140_vol"
   ScreenModuleView "Pump_FP_2" at 1181,795 size 243x168; ScreenModuleType ""
      Guid_{11997190-6812} <- "FP_Dtabase_Pump770A_visibility"
      Guid_{11997190-6818} <- "Pump770A_start"
      Guid_{11997190-6816} <- "Pump770A"
      Guid_{11997190-6820} <- "Pump770A_stop"
      Guid_{11997190-6822} <- "FP_Dtabase_Pump770A_tag_name"
   ScreenModuleView "Selenoid_FP_2" at 988,552 size 243x168; ScreenModuleType ""
      Guid_{11997190-6820} <- "SV1402_close"
      Guid_{11997190-6812} <- "FP_Dtabase_SV1402_visibility"
      Guid_{11997190-6818} <- "SV1402_open"
      Guid_{11997190-6816} <- "SV1402"
      Guid_{11997190-6822} <- "FP_Dtabase_SV1402_tag_name"
   ScreenModuleView "Selenoid_FP_1" at 483,551 size 243x168; ScreenModuleType ""
      Guid_{11997190-6820} <- "SV1401_close"
      Guid_{11997190-6812} <- "FP_Dtabase_SV1401_visibility"
      Guid_{11997190-6818} <- "SV1401_open"
      Guid_{11997190-6816} <- "SV1401"
      Guid_{11997190-6822} <- "FP_Dtabase_SV1401_tag_name"
   ScreenModuleView "Pump_FP_1" at 274,760 size 243x168; ScreenModuleType ""
      Guid_{11997190-6812} <- "FP_Dtabase_Pump100A_visibility"
      Guid_{11997190-6818} <- "Pump100A_start"
      Guid_{11997190-6816} <- "Pump100A"
      Guid_{11997190-6820} <- "Pump100A_stop"
      Guid_{11997190-6822} <- "FP_Dtabase_Pump100A_tag_name"

screen "Tank150" 1980x1078
   GraphicView "Graphic view_43" at 817,125 size 57x129; Picture "Graphic_19"
   GraphicView "Graphic view_10" at 721,189 size 251x329; Picture "Graphic_3"
   GraphicView "Graphic view_11" at 761,493 size 76x69; Picture "Graphic_4"
   GraphicView "Graphic view_12" at 772,556 size 83x93; Picture "Graphic_7"
   GraphicView "Graphic view_13" at 761,645 size 76x68; Picture "Graphic_4"
   GraphicView "Graphic view_14" at 854,494 size 76x69; Picture "Graphic_4"
   GraphicView "Graphic view_15" at 865,557 size 83x93; Picture "Graphic_7"
   GraphicView "Graphic view_16" at 854,641 size 76x177; Picture "Graphic_4"
   GraphicView "Graphic view_29" at 869,794 size 94x74; Picture "Graphic_14"
   GraphicView "Graphic view_28" at 736,706 size 87x74; Picture "Graphic_11"
   GraphicView "Graphic view_35" at 944,782 size 192x124; Picture "Graphic_16"
   GraphicView "Graphic view_26" at 560,732 size 192x124; Picture "Graphic_16"
      Appearance <- "Pump100A"
   Circle "Circle_1" at 628,771 size 48x48
      Appearance <- "Pump100A"
   Rectangle "Rectangle_3" at 787,575 size 23x56
      Appearance <- "SV1501"
   Rectangle "Rectangle_4" at 883,576 size 23x56
      Appearance <- "SV1502"
   Circle "Circle_2" at 1012,825 size 48x48
      Appearance <- "Pump770A"
   TextField "Text field_1" at 708,8 size 667x90; Text 'Tank 150'
   Group "Group_1" at 23,35 size 108x47
   Button "Button_5" at 1185,783 size 155x30; TextOff 'Pump770A FP'
      on Click: ResetBit("FP_Dtabase_Pump770A_visibility")
   Button "Button_4" at 992,540 size 155x30; TextOff 'SV1502 FP'
      on Click: ResetBit("FP_Dtabase_SV1502_visibility")
   Button "Button_2" at 487,539 size 155x30; TextOff 'SV1501 FP'
      on Click: ResetBit("FP_Dtabase_SV1501_visibility")
   Button "Button_6" at 278,764 size 155x30; TextOff 'Pump100A FP'
      on Click: ResetBit("FP_Dtabase_Pump100A_visibility")
   GraphicView "Graphic view_49" at 909,265 size 36x40; Picture "Graphic_20"
      Appearance <- "H_alarm_150"
   GraphicView "Graphic view_50" at 911,432 size 36x40; Picture "Graphic_21"
      Appearance <- "L_alarm_150"
   IOField "I/O field_1" at 894,127 size 117x51; FormatPattern 99999
      ProcessValue <- "Tank_150_cur_vol"
   Bar "Bar_1" at 826,238 size 42x271; MinimumValue 0; MaximumValue 100
      MinimumValue <- "my_variables_db_zero"
      MaximumValue <- "my_variables_db_tank_150_int_cap"
      ProcessValue <- "Tank_150_cur_vol"
   ScreenModuleView "Pump_FP_2" at 1181,777 size 243x168; ScreenModuleType ""
      Guid_{11997190-6822} <- "FP_Dtabase_Pump770A_tag_name"
      Guid_{11997190-6818} <- "Pump770A_start"
      Guid_{11997190-6816} <- "Pump770A"
      Guid_{11997190-6812} <- "FP_Dtabase_Pump770A_visibility"
      Guid_{11997190-6820} <- "Pump770A_stop"
   ScreenModuleView "Selenoid_FP_2" at 988,534 size 243x168; ScreenModuleType ""
      Guid_{11997190-6820} <- "SV1502_close"
      Guid_{11997190-6818} <- "SV1502_open"
      Guid_{11997190-6816} <- "SV1502"
      Guid_{11997190-6812} <- "FP_Dtabase_SV1502_visibility"
      Guid_{11997190-6822} <- "FP_Dtabase_SV1502_tag_name"
   ScreenModuleView "Selenoid_FP_1" at 483,533 size 243x168; ScreenModuleType ""
      Guid_{11997190-6820} <- "SV1501_close"
      Guid_{11997190-6818} <- "SV1501_open"
      Guid_{11997190-6816} <- "SV1501"
      Guid_{11997190-6812} <- "FP_Dtabase_SV1501_visibility"
      Guid_{11997190-6822} <- "FP_Dtabase_SV1501_tag_name"
   ScreenModuleView "Pump_FP_1" at 274,758 size 243x168; ScreenModuleType ""
      Guid_{11997190-6822} <- "FP_Dtabase_Pump100A_tag_name"
      Guid_{11997190-6818} <- "Pump100A_start"
      Guid_{11997190-6816} <- "Pump100A"
      Guid_{11997190-6812} <- "FP_Dtabase_Pump100A_visibility"
      Guid_{11997190-6820} <- "Pump100A_stop"
   Button "Button_1" at 63,53 size 68x12; TextOff 'Text'
      on Press: ActivateScreen("TankFarm", 0)

screen "Tank160" 1980x1078
   GraphicView "Graphic view_45" at 815,128 size 57x129; Picture "Graphic_19"
   GraphicView "Graphic view_19" at 721,192 size 251x329; Picture "Graphic_3"
   GraphicView "Graphic view_20" at 761,496 size 76x69; Picture "Graphic_4"
   GraphicView "Graphic view_21" at 772,559 size 83x93; Picture "Graphic_7"
   GraphicView "Graphic view_22" at 761,648 size 76x66; Picture "Graphic_4"
   GraphicView "Graphic view_23" at 854,497 size 76x69; Picture "Graphic_4"
   GraphicView "Graphic view_24" at 865,560 size 83x93; Picture "Graphic_7"
   GraphicView "Graphic view_28" at 736,707 size 87x74; Picture "Graphic_11"
   GraphicView "Graphic view_25" at 854,644 size 76x193; Picture "Graphic_4"
   GraphicView "Graphic view_36" at 869,820 size 94x74; Picture "Graphic_14"
   GraphicView "Graphic view_26" at 553,733 size 192x124; Picture "Graphic_16"
      Appearance <- "Pump100A"
   Circle "Circle_1" at 621,772 size 48x48
      Appearance <- "Pump100A"
   Rectangle "Rectangle_5" at 790,578 size 23x56
      Appearance <- "SV1601"
   Rectangle "Rectangle_6" at 884,579 size 23x56
      Appearance <- "SV1602"
   GraphicView "Graphic view_35" at 943,811 size 192x124; Picture "Graphic_16"
   Circle "Circle_2" at 1011,854 size 48x48
      Appearance <- "Pump770A"
   TextField "Text field_1" at 708,8 size 667x90; Text 'Tank 160'
   Group "Group" at 23,35 size 108x47
   Button "Button_5" at 1185,783 size 155x30; TextOff 'Pump770A FP'
      on Click: ResetBit("FP_Dtabase_Pump770A_visibility")
   Button "Button_4" at 992,540 size 155x30; TextOff 'SV1602 FP'
      on Click: ResetBit("FP_Dtabase_SV1602_visibility")
   Button "Button_2" at 487,539 size 155x30; TextOff 'SV1601 FP'
      on Click: ResetBit("FP_Dtabase_SV1601_visibility")
   Button "Button_6" at 278,748 size 155x30; TextOff 'Pump100A FP'
      on Click: ResetBit("FP_Dtabase_Pump100A_visibility")
   GraphicView "Graphic view_49" at 909,265 size 36x40; Picture "Graphic_20"
      Appearance <- "H_alarm_160"
   GraphicView "Graphic view_50" at 911,432 size 36x40; Picture "Graphic_21"
      Appearance <- "L_alarm_160"
   IOField "I/O field_1" at 894,127 size 117x51; FormatPattern 99999
      ProcessValue <- "Tank_160_cur_vol"
   Bar "Bar_1" at 826,241 size 42x271; MinimumValue 0; MaximumValue 100
      MinimumValue <- "my_variables_db_zero"
      ProcessValue <- "Tank_160_cur_vol"
      MaximumValue <- "my_variables_db_tank_160_int_cap"
   ScreenModuleView "Pump_FP_2" at 1181,777 size 243x168; ScreenModuleType ""
      Guid_{11997190-6822} <- "FP_Dtabase_Pump770A_tag_name"
      Guid_{11997190-6818} <- "Pump770A_start"
      Guid_{11997190-6816} <- "Pump770A"
      Guid_{11997190-6812} <- "FP_Dtabase_Pump770A_visibility"
      Guid_{11997190-6820} <- "Pump770A_stop"
   ScreenModuleView "Selenoid_FP_2" at 988,534 size 243x168; ScreenModuleType ""
      Guid_{11997190-6820} <- "SV1602_close"
      Guid_{11997190-6818} <- "SV1602_open"
      Guid_{11997190-6816} <- "SV1602"
      Guid_{11997190-6812} <- "FP_Dtabase_SV1602_visibility"
      Guid_{11997190-6822} <- "FP_Dtabase_SV1602_tag_name"
   ScreenModuleView "Selenoid_FP_1" at 483,533 size 243x168; ScreenModuleType ""
      Guid_{11997190-6820} <- "SV1601_close"
      Guid_{11997190-6818} <- "SV1601_open"
      Guid_{11997190-6816} <- "SV1601"
      Guid_{11997190-6812} <- "FP_Dtabase_SV1601_visibility"
      Guid_{11997190-6822} <- "FP_Dtabase_SV1601_tag_name"
   ScreenModuleView "Pump_FP_1" at 274,742 size 243x168; ScreenModuleType ""
      Guid_{11997190-6822} <- "FP_Dtabase_Pump100A_tag_name"
      Guid_{11997190-6818} <- "Pump100A_start"
      Guid_{11997190-6816} <- "Pump100A"
      Guid_{11997190-6812} <- "FP_Dtabase_Pump100A_visibility"
      Guid_{11997190-6820} <- "Pump100A_stop"
   Button "Button_1" at 63,53 size 68x12; TextOff 'Text'
      on Press: ActivateScreen("TankFarm", 0)

screen "Tank170" 1980x1078
   GraphicView "Graphic view_46" at 806,130 size 57x129; Picture "Graphic_19"
   GraphicView "Graphic view_41" at 676,188 size 327x414; Picture "Graphic_3"
   GraphicView "Graphic view_37" at 740,568 size 76x69; Picture "Graphic_4"
   GraphicView "Graphic view_38" at 751,631 size 83x93; Picture "Graphic_7"
   GraphicView "Graphic view_39" at 740,720 size 76x66; Picture "Graphic_4"
   GraphicView "Graphic view_40" at 715,779 size 87x74; Picture "Graphic_11"
   GraphicView "Graphic view_35" at 537,805 size 192x124; Picture "Graphic_16"
   GraphicView "Graphic view_32" at 861,568 size 76x69; Picture "Graphic_4"
   GraphicView "Graphic view_33" at 872,631 size 83x93; Picture "Graphic_7"
   GraphicView "Graphic view_34" at 861,716 size 76x177; Picture "Graphic_4"
   GraphicView "Graphic view_36" at 877,877 size 94x74; Picture "Graphic_14"
   GraphicView "Graphic view_42" at 959,868 size 192x124; Picture "Graphic_16"
   Rectangle "Rectangle_7" at 768,650 size 23x56
      Appearance <- "SV1701"
   Rectangle "Rectangle_8" at 889,650 size 23x56
      Appearance <- "SV1702"
   Circle "Circle_2" at 605,848 size 48x48
      Appearance <- "Pump770A"
   Circle "Circle_3" at 1028,909 size 48x48
      Appearance <- "Pump771A"
   TextField "Text field_1" at 708,8 size 665x90; Text 'Tank 170'
   Group "Group" at 23,35 size 108x47
   Button "Button_5" at 1191,859 size 155x30; TextOff 'Pump771A FP'
      on Click: ResetBit("FP_Dtabase_Pump771A_visibility")
   Button "Button_4" at 982,619 size 155x30; TextOff 'SV1702 FP'
      on Click: ResetBit("FP_Dtabase_SV1702_visibility")
   Button "Button_2" at 461,624 size 155x30; TextOff 'SV1701 FP'
      on Click: ResetBit("FP_Dtabase_SV1701_visibility")
   Button "Button_6" at 278,828 size 155x30; TextOff 'Pump770A FP'
      on Click: ResetBit("FP_Dtabase_Pump770A_visibility")
   GraphicView "Graphic view_53" at 905,272 size 36x40; Picture "Graphic_20"
      Appearance <- "H_alarm_170"
   GraphicView "Graphic view_54" at 907,507 size 36x40; Picture "Graphic_21"
      Appearance <- "L_alarm_170"
   IOField "I/O field_4" at 890,134 size 117x51; FormatPattern 99999
      ProcessValue <- "Tank_170_cur_vol"
   Bar "Bar_4" at 813,224 size 56x366; MinimumValue 0; MaximumValue 100
      MinimumValue <- "my_variables_db_zero"
      ProcessValue <- "Tank_170_cur_vol"
      MaximumValue <- "my_variables_db_tank_170_int_cap"
   ScreenModuleView "Pump_FP_2" at 1187,853 size 243x168; ScreenModuleType ""
      Guid_{11997190-6818} <- "Pump771A_start"
      Guid_{11997190-6816} <- "Pump771A"
      Guid_{11997190-6820} <- "Pump771A_stop"
      Guid_{11997190-6812} <- "FP_Dtabase_Pump771A_visibility"
      Guid_{11997190-6822} <- "FP_Dtabase_Pump771A_tag_name"
   ScreenModuleView "Selenoid_FP_2" at 978,613 size 243x168; ScreenModuleType ""
      Guid_{11997190-6820} <- "SV1702_close"
      Guid_{11997190-6818} <- "SV1702_open"
      Guid_{11997190-6816} <- "SV1702"
      Guid_{11997190-6812} <- "FP_Dtabase_SV1702_visibility"
      Guid_{11997190-6822} <- "FP_Dtabase_SV1702_tag_name"
   ScreenModuleView "Selenoid_FP_1" at 457,618 size 243x168; ScreenModuleType ""
      Guid_{11997190-6820} <- "SV1701_close"
      Guid_{11997190-6818} <- "SV1701_open"
      Guid_{11997190-6816} <- "SV1701"
      Guid_{11997190-6812} <- "FP_Dtabase_SV1701_visibility"
      Guid_{11997190-6822} <- "FP_Dtabase_SV1701_tag_name"
   ScreenModuleView "Pump_FP_1" at 274,822 size 243x168; ScreenModuleType ""
      Guid_{11997190-6812} <- "FP_Dtabase_Pump770A_visibility"
      Guid_{11997190-6818} <- "Pump770A_start"
      Guid_{11997190-6816} <- "Pump770A"
      Guid_{11997190-6820} <- "Pump770A_stop"
      Guid_{11997190-6822} <- "FP_Dtabase_Pump770A_tag_name"
   Button "Button_1" at 63,53 size 68x12; TextOff 'Text'
      on Press: ActivateScreen("TankFarm", 0)

screen "AlarmScreen" 1980x1078
   AlarmView "Alarm view_1" at 163,167 size 1566x825
   Group "Group" at 25,36 size 108x47
   TextField "Text field_1" at 637,13 size 877x90; Text 'Alarm Screen'
   Button "Button_1" at 65,54 size 68x12; TextOff 'Text'
      on Press: ActivateScreen("TankFarm", 0)

PopupScreen "lo_alarm_pop_up" 300x240
   TextField "Text field_1" at 14,10 size 235x22; Text 'Low Level Occured'
   TextField "Text field_5" at 15,138 size 224x22; Text 'Corrective Actions:'
   TextField "Text field_6" at 15,162 size 152x20; Text 'Open inlet valve'
   TextField "Text field_7" at 15,82 size 260x22; Text 'Consequence of no Action:'
   TextField "Text field_8" at 15,105 size 136x19; Text 'Empty Tank'
   Button "Button_2" at 269,6 size 22x28; TextOff 'X'
      on Click: function_efd93a16("lo_alarm_pop_up", 0, 0, 0, -1, 1)

PopupScreen "hi_alarm_pop_up" 300x240
   Button "Button_2" at 269,6 size 22x28; TextOff 'X'
      on Click: function_efd93a16("hi_alarm_pop_up", 0, 0, 0, -1, 1)
   TextField "Text field_1" at 14,10 size 238x22; Text 'High Level Occured'
   TextField "Text field_5" at 15,138 size 224x22; Text 'Corrective Actions:'
   TextField "Text field_6" at 15,162 size 208x20; Text 'Close inlet valve'
   TextField "Text field_7" at 15,82 size 260x22; Text 'Consequence of no Action:'
   TextField "Text field_8" at 15,105 size 224x19; Text 'Overfill and overpressure'

screen "Trend Screen" 1980x1078
   TrendView "Trend view_1" at 67,159 size 1722x883
   TextField "Text field_1" at 641,8 size 866x90; Text 'Trend Screen'
   Group "Group" at 23,35 size 108x47
   Button "Button_1" at 63,53 size 68x12; TextOff 'Text'
      on Press: ActivateScreen("TankFarm", 0)

scheduled task "ChangeUserTask"
   on Action: function_f41c6f6c("Current_user"); function_de9337da(); function_e1ab61de("current_group_no")
*)

(* ===== HMI "HMI_RT_1" =====
system functions are stored by id; their names below are inferred from use

HMI tags "Default tag table"
   "Pump_fp_visibility" : Bool, internal

text list "Status": 0 'Closed'; 1 'Opened'

ScreenModuleEditorView "Selenoid_FP" 640x480
   Rectangle "Rectangle_3" at 10,10 size 243x168
      Visibility <- "SV_fp_visibility_"
   Button "Button_2" at 222,17 size 22x28; TextOff 'X'
      on Click: SetBit("SV_fp_visibility_")
      ProcessValue <- "SV_fp_visibility_"
      Visibility <- "SV_fp_visibility_"
   Line "Line_1" at 12,47 size 239x0
      Visibility <- "SV_fp_visibility_"
   Button "Button_4" at 140,138 size 91x28; TextOff 'Open'
      on Release: ResetBit("SV_open")
      on Press: SetBit("SV_open")
      Visibility <- "SV_fp_visibility_"
      ProcessValue <- "SV_open"
   Line "Line_2" at 12,131 size 239x0
      Visibility <- "SV_fp_visibility_"
   Button "Button_3" at 27,138 size 89x28; TextOff 'Close'
      on Release: ResetBit("SV_close")
      on Press: SetBit("SV_close")
      Visibility <- "SV_fp_visibility_"
      ProcessValue <- "SV_close"
   Line "Line_3" at 125,132 size 0x44
      Visibility <- "SV_fp_visibility_"
   IOField "I/O field_1" at 21,18 size 140x25; FormatPattern ???????????????
      Visibility <- "SV_fp_visibility_"
      ProcessValue <- "SV_tag_name"
   TextField "Text field_2" at 11,73 size 88x24; Text 'Status :'
      Visibility <- "SV_fp_visibility_"
   SymbolicIOField "Symbolic I/O field_1" at 90,71 size 116x32; TextOn '1'; TextOff '0'; TextList "Status"
      Visibility <- "SV_fp_visibility_"
      ProcessValue <- "SV_stat"
*)

(* ===== HMI "HMI_RT_1" =====
system functions are stored by id; their names below are inferred from use

HMI tags "Default tag table"
   "Pump_fp_visibility" : Bool, internal

text list "Status": 0 'OFF'; 1 'ON'

ScreenModuleEditorView "Pump_FP" 640x480
   Rectangle "Rectangle_3" at 10,10 size 243x168
      Visibility <- "Pump_fp_visibility_"
   Button "Button_2" at 222,17 size 22x28; TextOff 'X'
      on Click: SetBit("Pump_fp_visibility_")
      ProcessValue <- "Pump_fp_visibility_"
      Visibility <- "Pump_fp_visibility_"
   Line "Line_1" at 12,47 size 239x0
      Visibility <- "Pump_fp_visibility_"
   Button "Button_4" at 140,138 size 91x28; TextOff 'Start'
      on Release: ResetBit("Pump_start")
      on Press: SetBit("Pump_start")
      Visibility <- "Pump_fp_visibility_"
      ProcessValue <- "Pump_start"
   Line "Line_2" at 12,131 size 239x0
      Visibility <- "Pump_fp_visibility_"
   Button "Button_3" at 27,138 size 89x28; TextOff 'Stop'
      on Release: ResetBit("Pump_stop")
      on Press: SetBit("Pump_stop")
      Visibility <- "Pump_fp_visibility_"
      ProcessValue <- "Pump_stop"
   Line "Line_3" at 125,132 size 0x44
      Visibility <- "Pump_fp_visibility_"
   IOField "I/O field_1" at 21,18 size 140x25; FormatPattern ???????????????
      Visibility <- "Pump_fp_visibility_"
      ProcessValue <- "Pump_tag_name"
   TextField "Text field_2" at 11,73 size 88x24; Text 'Status :'
      Visibility <- "Pump_fp_visibility_"
   SymbolicIOField "Symbolic I/O field_1" at 90,71 size 96x32; TextOn '1'; TextOff '0'; TextList "Status"
      Visibility <- "Pump_fp_visibility_"
      ProcessValue <- "Pump_stat"
*)